{attribute 'TcGenerated'}
{attribute 'no-analysis'}
{attribute 'linkalways'}
// This function has been automatically generated from the project information.
VAR_GLOBAL CONSTANT
	{attribute 'const_non_replaced'}
	stLibVersion_Base_Library : ST_LibVersion := (iMajor := 3, iMinor := 1, iBuild := 0, iRevision := 0, nFlags := 0, sVersion := '3.1.0.0');
END_VAR

(* stored: Version 1.1.0.1
   GVL Global_Version: Id {acf6c8a9-288a-49ea-9b98-dd493e021fb0} *)
